// TwinCAT 3 PLC project lamp_motion
// Title: tmo_lamp_motion
// Company: SLAC
// ProjectVersion: 1.0.4
// ProgramVersion: 3.1.4022.7
// libraries:
//   Tc2_MC2, * (Beckhoff Automation GmbH)
//   Tc2_Standard, * (Beckhoff Automation GmbH)
//   Tc2_System, * (Beckhoff Automation GmbH)
//   Tc2_Utilities, * (Beckhoff Automation GmbH)
//   Tc3_Module, * (Beckhoff Automation GmbH)
//   lcls-twincat-motion,1.8.0,SLAC
// project tree:
//   / PlcTask.TcTTO (not stored)
//   Version/ Global_Version.TcGVL
//   POUs/ Main.TcPOU (not stored)

// ---- Version/Global_Version.TcGVL
{attribute 'TcGenerated'}
// This function has been automatically generated from the project information.
VAR_GLOBAL CONSTANT
    {attribute 'const_non_replaced'}
    {attribute 'linkalways'}
    stLibVersion_tmo_lamp_motion : ST_LibVersion := (iMajor := 1, iMinor := 0, iBuild := 4, iRevision := 0, sVersion := '1.0.4');
END_VAR
